{attribute 'qualified_only'}
{attribute 'strict'}
{attribute 'to_string'}
/// Enum ***DUT***
TYPE DUT :
(
	member1 := 0, //< default
	member2 := 10, //< nr 10
	meber3 := 20, //< nr 20
	meber4 := 30 //< nr 30
);
END_TYPE
//  meber4 = '30 '

(* stored: Version 1.1.0.1
   EnumerationTextList DUT: Id {d2b065b2-0a82-4fb0-8aa5-405ff1674b3c} *)
